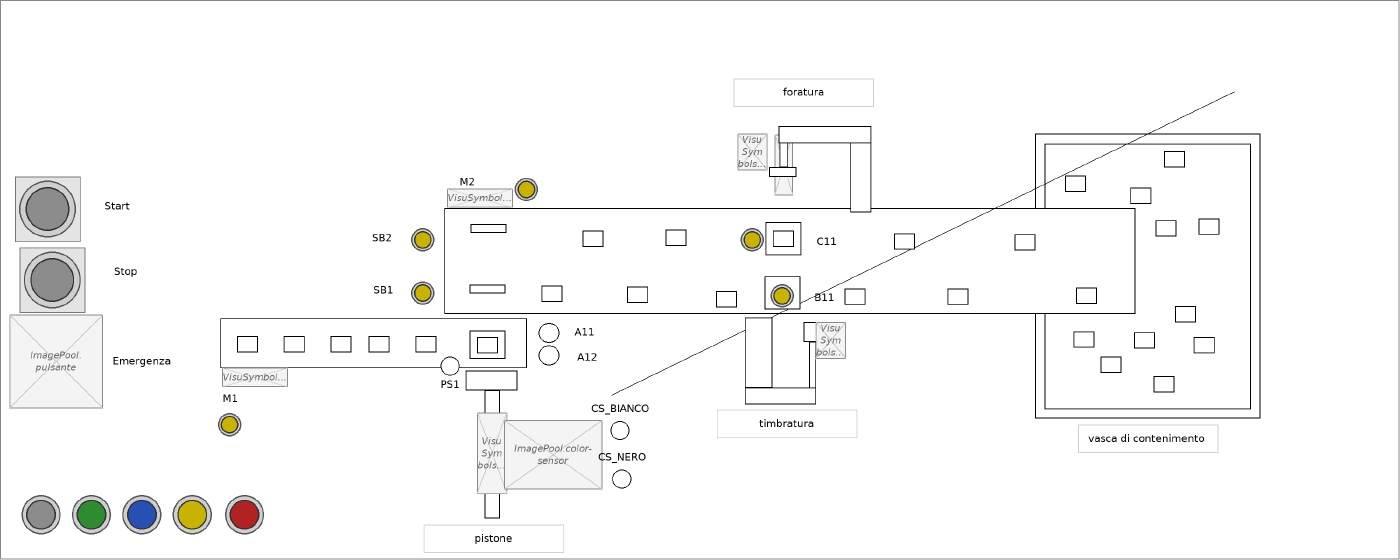
VISUALIZATION Visualization  // 1500x600
    PushSwitch (16,189 70x70), variable: GVL.PB1, behaviour: TAP, style: Switch-PushSwitch-Gray
    Label (98,206 55x30), "Start"
    PushSwitch (21,265 70x70), variable: GVL.PB2, behaviour: TAP, style: Switch-PushSwitch-Gray
    Label (102,276 65x30), "Stop"
    Label (107,372 90x30), "Emergenza"
    Lamp1 (20,527 48x49), variable: GVL.L1, style: Lamp-Lamp1-Gray
    Lamp1 (74,527 48x49), variable: GVL.L2, style: Lamp-Lamp1-Green
    Lamp1 (128,527 48x49), variable: GVL.L3, style: Lamp-Lamp1-Blue
    Lamp1 (182,527 48x49), variable: GVL.L4, style: Lamp-Lamp1-Yellow
    Lamp1 (238,527 48x49), variable: GVL.L5, style: Lamp-Lamp1-Red
    Image (10,337 100x100), image: ImagePool.pulsante
        OnMouseClick: toggle GVL.PBE
    Textfield (454,562 150x30), "pistone"
    Image (830,144 19x65), image: VisuSymbols.Symbols.ArrowBoldDown
    RoundedRectangle (1109,143 241x305)
    RoundedRectangle (1119,154 221x284)
    Rectangle (236,341 328x53)
    RoundedRectangle (476,223 740x113)
    Line (655,423) (1322,98)
    RoundedRectangle (499,397 55x21)
    Rectangle (519,418 16x137)
    Image (511,442 32x87), image: VisuSymbols.Symbols.DoubleArrow4
    Rectangle (254,360 22x17)
    Rectangle (304,360 22x17)
    Rectangle (354,360 22x17)
    Rectangle (395,360 22x17)
    Rectangle (624,247 22x17)
    Rectangle (713,246 22x17)
    Rectangle (445,360 22x17)
    Rectangle (580,306 22x17)
    Rectangle (672,307 22x17)
    Rectangle (767,312 22x17)
    Rectangle (905,309 22x17)
    Rectangle (1015,309 22x17)
    Rectangle (1153,308 22x17)
    Rectangle (958,250 22x17)
    Rectangle (1087,251 22x17)
    Rectangle (1179,382 22x17)
    Rectangle (1279,361 22x17)
    Rectangle (1259,328 22x17)
    Rectangle (1215,356 22x17)
    Rectangle (1150,355 22x17)
    Rectangle (1236,403 22x17)
    Rectangle (1141,188 22x17)
    Rectangle (1211,201 22x17)
    Rectangle (1247,162 22x17)
    Rectangle (1238,236 22x17)
    Rectangle (1284,234 22x17)
    Textfield (1155,455 150x30), "vasca di contenimento"
    RoundedRectangle (861,345 19x21)
    Rectangle (867,366 7x51)
    Rectangle (798,415 76x18)
    Rectangle (798,340 29x75)
    Image (874,345 32x39), image: VisuSymbols.Symbols.DoubleArrow4
    Textfield (768,439 150x30), "timbratura"
    Textfield (786,84 150x30), "foratura"
    Rectangle (911,152 22x75)
    RoundedRectangle (824,179 29x10)
    Rectangle (835,150 9x29)
    Rectangle (834,135 99x18)
    Image (790,143 32x39), image: VisuSymbols.Symbols.DoubleArrow4
    Image (479,202 70x20), image: VisuSymbols.Symbols.ArrowBoldRight
    Image (238,394 70x20), image: VisuSymbols.Symbols.ArrowBoldRight
    Rectangle (503,354 38x30)
    Rectangle (511,361 22x17)
    Rectangle (820,238 38x35)
    Rectangle (819,296 38x35)
    Rectangle (828,247 22x17)
    Rectangle (504,240 38x9)
    Rectangle (503,305 38x9)
    Lamp1 (439,242 28x30), variable: MAIN.SB2, style: Lamp-Lamp1-Yellow
    Lamp1 (439,299 28x30), variable: MAIN.SB1, style: Lamp-Lamp1-Yellow
    Lamp1 (824,302 28x30), variable: MAIN.B1, style: Lamp-Lamp1-Yellow
    Lamp1 (792,242 28x30), variable: MAIN.C1, style: Lamp-Lamp1-Yellow
    Label (205,412 84x30), "M1"
    Label (459,180 84x30), "M2"
    Label (600,341 53x30), "A11"
    Label (858,244 56x30), "C11"
    Label (605,368 49x30), "A12"
    Label (388,296 46x30), "SB1"
    Label (385,240 49x30), "SB2"
    Label (855,304 57x30), "B11"
    Ellipse (577,346 22x21)
        tap MAIN.A11
    Ellipse (577,370 22x21)
        tap MAIN.A12
    Lamp1 (232,440 28x30), variable: MAIN.motore1, style: Lamp-Lamp1-Yellow
    Lamp1 (550,188 28x30), variable: MAIN.motore2, style: Lamp-Lamp1-Yellow
    Ellipse (654,451 20x20), colour toggle: GVL.M1
    Label (622,432 85x12), "CS_BIANCO"
    Ellipse (472,382 20x20), colour toggle: GVL.M1
    Label (463,406 39x12), "PS1"
    Image (540,450 105x74), image: ImagePool.color-sensor
    Ellipse (656,503 20x20), colour toggle: GVL.M1
    Label (624,484 85x12), "CS_NERO"
END_VISUALIZATION

(* stored: Version 1.1.0.1, ProductVersion 3.1.4024.12
   Visu Visualization: Id {e3399594-b7fd-4589-9a49-3967da9e8e84} *)
